{attribute 'no_explicit_call' := 'direct call for this function block is not allowed'}
FUNCTION_BLOCK FB_MathMachine
VAR
	_nValue : DINT;
END_VAR

{attribute 'TcRpcEnable'}
METHOD DivideValues : DINT
VAR_INPUT
	nNumerator, 
	nDenominator : DINT;
END_VAR
VAR_OUTPUT
	nRemainder   : DINT;
END_VAR
IF nDenominator <> 0 THEN
	DivideValues := nNumerator / nDenominator;
	nRemainder   := nNumerator MOD nDenominator;
END_IF
END_METHOD

{attribute 'TcRpcEnable'}
METHOD GetValue : DINT
VAR_INPUT
END_VAR
GetValue := THIS^._nValue;
END_METHOD

{attribute 'TcRpcEnable'}
METHOD Reset
VAR_INPUT
END_VAR
 THIS^._nValue := 0;
END_METHOD

{attribute 'TcRpcEnable'}
METHOD SetValue
VAR_INPUT
	nValue : DINT;
END_VAR
THIS^._nValue := nValue;
END_METHOD

{attribute 'TcRpcEnable'}
METHOD SumValues : DINT
VAR_INPUT
	nValue1, nValue2 : DINT;
END_VAR
SumValues := nValue1 + nValue2;
END_METHOD

END_FUNCTION_BLOCK

(* stored: Version 1.1.0.1, ProductVersion 3.1.4024.15
   POU FB_MathMachine: Id {bb1278ac-4e17-40b6-8919-426e05c4676c}, SpecialFunc None
   Method DivideValues: Id {b33507e4-e5b5-4046-ba42-b67bce270c2e}
   Method GetValue: Id {93b38f2b-0b4e-4a95-a0bb-8f5035ef869e}
   Method Reset: Id {d1c73aae-7c11-4a69-9422-86211b8b5102}
   Method SetValue: Id {1540aca3-3be9-4d9f-9e83-8166da4e56ca}
   Method SumValues: Id {e74e39bd-9ed2-4049-988d-b3509be6be4b} *)
